# EPICS substitutions: db/PSI/ecmcILK_v2.substitutions
file "ecmcEcSlave.template"
{
  pattern {}
          {}
}

file "ecmcILK_v2.template"
{
  pattern {CH_ID, DTYP,              FTVL ,  KEY,        }
          {01,    "asynInt8ArrayIn", "CHAR", "byteOutputBuff"  }
          {02,    "asynInt8ArrayIn", "CHAR", "byteInputBuff" }
}
